(*udt (user defined type) of Beckhoff EL2624 - 4 Point Relay Type Output Terminal:
	Auth: j.vandongen
	October 2019*)


TYPE udt_EP2624 :
STRUCT
	Q: INT;
END_STRUCT
END_TYPE

(* stored: Version 1.1.0.1, ProductVersion 3.1.4024.9
   DUT udt_EP2624: Id {516404b0-ca6e-40ba-b569-04002fa3fced} *)
